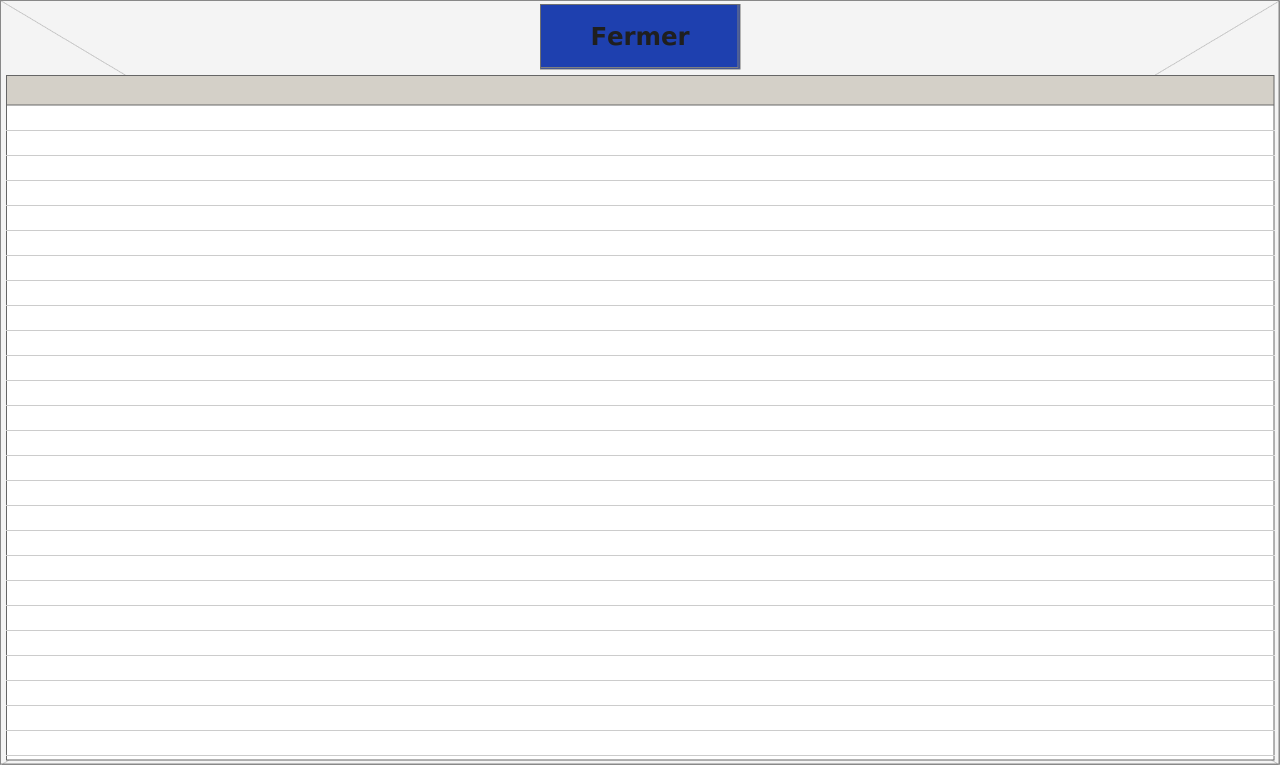
VISUALIZATION Alarmes  // 1280x765
    Image (0,0 1280x765), image: ImagePool.Fond_Degr
    Button (540,4 200x65), "Fermer"
        OnMouseDown: CloseDialog Dialog=Alarmes, Result=OK, NumpadKeypadSet=True
    Table (6,75 1268x685), invisible if: VisuElems.CURRENTLANGUAGE = 'en', data array: Alarmes.Tab_Alarme_FREN
        p3854506369: Alarmes.Tab_Alarme_FREN[1,INDEX]
        p1892666644: Alarmes.Tab_Alarme_FREN[2,INDEX]
    Table (6,75 1268x685), invisible if: VisuElems.CURRENTLANGUAGE = 'fr', data array: Alarmes.Tab_Alarme_FREN
        p3854506369: Alarmes.Tab_Alarme_FREN[1,INDEX]
        p1892666644: Alarmes.Tab_Alarme_FREN[2,INDEX]
END_VISUALIZATION

(* stored: Version 1.1.0.1, ProductVersion 3.1.4024.15
   Visu Alarmes: Id {3639146b-d6dc-44b8-a843-80ed3aac3bfe} *)
